(* CoDeSys 2.3 library: TcTestAndSet.lib *)
(* Libraries: STANDARD.LIB 5.6.98 09:45:02 *)

(* POU TestAndSet, ST *)
FUNCTION TestAndSet : BOOL
VAR_IN_OUT
	Flag	:	BOOL; (* Flag to check if TRUE or FALSE *)
END_VAR
;
END_FUNCTION
